(*********************************** G.D S.p.A. - Technical Department ***********************************
============= PROGRAM INFO ============
FOLDER:             TBD
MACHINES INVOLVED:  TBD 

============= DESCRIPTION =============
csp machine declaration

============= REVISIONS ===============
Date		Version	 	Author      	Description             
----------	-------		------------  	--------------------------------------------
2019/04/05 	0000.00	 	M.Grasso		Creation of the PRG

**********************************************************************************************************)
(*$R process_ref := prc; $*)
PROGRAM csp_case_topRail_accU
VAR
	
	prc:											process;
	prc_path:										STRING;
	
END_VAR

_read_var_input();

_object_manager();

IF NOT objects_running()
THEN
	RETURN;	
END_IF

_read_process_image();

_mode_manager();

_set_runtime_properties();

(********************************* BODY *********************************)
(************************************************************************)

_handle_messages();

_write_output();

ACTION _handle_messages:
;
END_ACTION

ACTION _handle_process_test:
;
END_ACTION

ACTION _mode_manager:
IF process_mode_req_is_pending(prc)
THEN
    process_apply_mode_req_first_step(prc);
    CASE process_get_mode(prc) OF
        MODE_TO_ABSENT:
			;
        MODE_TO_INACTIVE:
			;
        MODE_TO_TEST:
			;
        MODE_TO_OPERATIONAL:
			;
    END_CASE
    process_apply_mode_req_second_step(prc);
END_IF
END_ACTION

ACTION _object_manager:
IF objects_initialization()
THEN
	sub_process_init(
		object_name					:= 'csp_case_topRail_accU.prc', 
		process						:= csp_case_topRail.prc, 
		CONVERSION_this				:= prc);
		
	prc_path 						:= process_get_path(prc);
END_IF

IF objects_running()
THEN
	process_cycle(prc);
END_IF
END_ACTION

ACTION _read_process_image:
;
END_ACTION

ACTION _read_var_input:
;
END_ACTION

ACTION _set_runtime_properties:
;
END_ACTION

ACTION _write_output:
;
END_ACTION

END_PROGRAM

(* stored: Version 1.1.0.1, ProductVersion 3.1.4022.12
   POU csp_case_topRail_accU: Id {f64c0f9f-43e7-4fbe-9400-b9213006544e}, SpecialFunc None
   Action _handle_messages: Id {e7d13a5d-9414-44a0-ac8f-b8923ae88d0d}
   Action _handle_process_test: Id {56d7a084-f148-4607-88fe-8217df3ac7bf}
   Action _mode_manager: Id {94e04fd7-aefa-41c6-befe-259b4297e877}
   Action _object_manager: Id {cc9c5f18-66a3-43dd-aece-a4c9c46a6f65}
   Action _read_process_image: Id {b719cfba-0612-4b6d-84db-d43592a1b0ac}
   Action _read_var_input: Id {3572bb9f-9250-4def-8a4a-fb8b54015195}
   Action _set_runtime_properties: Id {9c555fd3-f13c-494b-9e98-48167448307d}
   Action _write_output: Id {3ceaeceb-2583-4d7b-9ff5-0260097da993} *)
